ABB RobotStudio station: RemoteControlledYumi.rspag

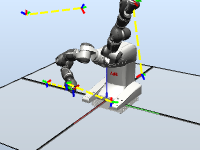
--- station ---
Station RemoteControlledYumi (saved by RobotStudio 6.5.7496.1049)
Controller IRB_14000_0.5kg_0.5m
  mechanical unit ROB_R: IRB14000_0.5_0.5_R, 6 joints, base frame (0, 0, 0) mm
  mechanical unit ROB_R_7: IRB14000_0.5_0.5_R, 1 joints, base frame (0, 0, 0) mm
  mechanical unit ROB_L: IRB14000_0.5_0.5_L, 6 joints, base frame (0, 0, 0) mm
  mechanical unit ROB_L_7: IRB14000_0.5_0.5_L, 1 joints, base frame (0, 0, 0) mm
Layout (positions relative to the parent item):
  - IRB14000_0.5_0.5 [mechanism, from Robots\IRB14000_0.5_0.5__01.rslib] at (0, 0, 0) mm
  - IRB14000_0.5_0.5_R [mechanism, from Robots\IRB14000_0.5_0.5__01.rslib] at (0, 0, 0) mm; joint values [1.0888, -1.6327, -1.6401, 0.7242, 2.6336, 0.3087, -2.7827] (rad or m)
  - IRB14000_0.5_0.5_L [mechanism, from Robots\IRB14000_0.5_0.5__01.rslib] at (0, 0, 0) mm; joint values [0.5159, -0.7237, 1.0056, -1.384, 2.6336, 0.3087, -2.7827] (rad or m)

--- Backups/IRB_14000_0.5kg_0.5m/RAPID/TASK1/PROGMOD/Module1.mod ---
MODULE Module1
	CONST jointtarget JointTarget_3:=[[5.435483871,-60.25483871,20.919354839,150.895790314,17.687340054,-159.437228739],[57.616129032,9E+09,9E+09,9E+09,9E+09,9E+09]];
	CONST jointtarget JointTarget_4:=[[29.560965021,-41.462551121,-79.294754901,150.895790314,17.687340054,-159.437228739],[57.616129032,9E+09,9E+09,9E+09,9E+09,9E+09]];
	CONST jointtarget JointTarget_1:=[[44.570967742,-88.003225806,2.538709677,0,39.999998836,0],[-79.358064516,9E+09,9E+09,9E+09,9E+09,9E+09]];
	CONST jointtarget JointTarget_2:=[[62.386456105,-93.54618891,41.493211378,150.895790314,17.687340054,-159.437228739],[-93.969401092,9E+09,9E+09,9E+09,9E+09,9E+09]];

    PROC main()
        RunLoop;
    ENDPROC
	PROC wavehigh()
	    MoveAbsJ JointTarget_3,v1000,fine,tool0\WObj:=wobj0;
	    MoveAbsJ JointTarget_4,v1000,z100,tool0\WObj:=wobj0;
	ENDPROC
	PROC wavelow()
	    MoveAbsJ JointTarget_1,v1000,z100,tool0\WObj:=wobj0;
	    MoveAbsJ JointTarget_2,v1000,z100,tool0\WObj:=wobj0;
	ENDPROC
ENDMODULE

--- Backups/IRB_14000_0.5kg_0.5m/RAPID/TASK1/PROGMOD/Remote.mod ---
MODULE Remote
    TASK PERS bool start := FALSE;
    TASK PERS bool running := FALSE;

    TASK PERS string name := "wavelow";

    PROC Init()
        start := FALSE;
        running := FALSE;
    ENDPROC

    PROC RunLoop()
        Init;
        WHILE TRUE DO
            WHILE NOT start DO
                WaitTime .1;
            ENDWHILE
            start := FALSE;
            running := TRUE;
            %name%;
            running := FALSE;
        ENDWHILE
    ENDPROC
ENDMODULE

--- Backups/IRB_14000_0.5kg_0.5m/RAPID/TASK1/SYSMOD/LINKEDM.sys ---
%%%
  VERSION:1
  LANGUAGE:ENGLISH
%%%

MODULE LINKEDM (SYSMODULE)

! FOLLOWER
!     Name of electronically linked follower axis used by operator at teach pendent.
      PERS string l_f_axis_name{5}       :=  ["",  "", "", "", ""];

!     Name of the mechanical unit for follower axis.
      PERS string l_f_mecunt_n{5}  :=  ["", "", "", "", ""];

!     Linked follower axis number in the mechanical unit (first axis in mech. unit is number 1).
      PERS num l_f_axis_no{5}      :=  [0,          0,   0,  0,  0];

! MASTER
!     Name of the mechanical unit for linked master axis.
      PERS string l_m_mecunt_n{5} :=  ["", "", "", "", ""];

!     Linked master axis number in the mechanical unit (first axis in mech. unit is number 1).
!     See axis number table in documentation for different master mechanical units.
      PERS num l_m_axis_no{5}     :=  [0,  0,  0,  0,  0];

! POSITION OFFSET
!     The increase of the allowed offset position between the master and follower
!     positions, used when starting AUTO mode. As soon as the offset is decreased
!     the old configurated parameter is used.
!     Example: 3 => the configurated value of allowed offset is increased 3 times.
      PERS num offset_ratio{5}       :=  [10,  10,   10,  10,  10];

! SPEED RATIO
!     Speed_ratio used in AUTO and JOG modes [ very_slow   slow    normal    fast]
!     Value 1 = max allowed manual speed.
      CONST num speed_ratio {20}      := [0.01, 0.01, 0.01, 0.01, 0.01,
                                          0.05, 0.05, 0.05, 0.05, 0.05,
                                          0.20, 0.20, 0.20, 0.20, 0.20,
                                          1.00, 1.00, 1.00, 1.00, 1.00];

! STEP SIZE
!     Displacement position used in JOG mode for each activation of positive or
!     negative movement.                  [very_short    short   normal   long]
!     Unit degees or meter.
      CONST num displacement {20}     := [0.001, 0.001, 0.001, 0.001, 0.001,
                                          0.005, 0.005, 0.005, 0.005, 0.005,
                                          0.020, 0.020, 0.020, 0.020, 0.020,
                                          0.100, 0.100, 0.100, 0.100, 0.100];


!-------------------------------------------------------------
 PROC Linked_m ()
      Linked_m_exe ;
 ENDPROC
ENDMODULE

--- Backups/IRB_14000_0.5kg_0.5m/RAPID/TASK2/PROGMOD/Module1.mod ---
MODULE Module1
	CONST jointtarget JointTarget_3:=[[5.435483871,-60.25483871,20.919354839,150.895790314,17.687340054,-159.437228739],[57.616129032,9E+09,9E+09,9E+09,9E+09,9E+09]];
	CONST jointtarget JointTarget_4:=[[29.560965021,-41.462551121,-79.294754901,150.895790314,17.687340054,-159.437228739],[57.616129032,9E+09,9E+09,9E+09,9E+09,9E+09]];
	CONST jointtarget JointTarget_1:=[[132.81046026,22.322183296,1.519468535,17.333519179,42.225247147,-11.8465977],[-86.991502251,9E+09,9E+09,9E+09,9E+09,9E+09]];
	CONST jointtarget JointTarget_2:=[[132.81046026,-30.727265036,-31.120707126,17.333519179,42.225247147,-11.8465977],[-86.991502251,9E+09,9E+09,9E+09,9E+09,9E+09]];

    PROC main()
        RunLoop;
    ENDPROC

	PROC wavehigh()
	    MoveAbsJ JointTarget_3,v1000,z100,tool0\WObj:=wobj0;
	    MoveAbsJ JointTarget_4,v1000,z100,tool0\WObj:=wobj0;
	ENDPROC

	PROC wavelow()
	    MoveAbsJ JointTarget_1,v1000,z100,tool0\WObj:=wobj0;
	    MoveAbsJ JointTarget_2,v1000,z100,tool0\WObj:=wobj0;
	ENDPROC
ENDMODULE

--- Backups/IRB_14000_0.5kg_0.5m/RAPID/TASK2/PROGMOD/Remote.mod ---
MODULE Remote
    TASK PERS bool start := FALSE;
    TASK PERS bool running := FALSE;

    TASK PERS string name := "wavehigh";

    PROC Init()
        start := FALSE;
        running := FALSE;
    ENDPROC

    PROC RunLoop()
        Init;
        WHILE TRUE DO
            WHILE NOT start DO
                WaitTime .1;
            ENDWHILE
            start := FALSE;
            running := TRUE;
            %name%;
            running := FALSE;
        ENDWHILE
    ENDPROC
ENDMODULE

--- Backups/IRB_14000_0.5kg_0.5m/SYSPAR/EIO.cfg ---
EIO:CFG_1.0:6:1::
#
SYSSIG_IN:

      -Signal "Collision_Avoidance" -Action "CollAvoidance"
#
INDUSTRIAL_NETWORK:

      -Name "EtherNetIP" -Connection "Private Network"\
      -Label "EtherNet/IP Adapter Network"

      -Name "DeviceNet" -Label "DeviceNet Master/Slave Network" -Address "2"
#
EIO_CROSS:

      -Name "Cross_Signal_Lamp" -Res "Signal_Lamp" -Act1 "DRV1BRAKE"
#
EIO_SIGNAL_SAFELEVEL:

      -Name "FlangePowerSafeLevel" -ActionWhenStartup "Last"
#
DEVICENET_DEVICE:

      -Name "D652_10" -VendorName "ABB Robotics" -ProductName "24 VDC Unit"\
      -Address 10 -ProductCode 26 -DeviceType 7 -ConnectionType "COS"\
      -OutputSize 2 -InputSize 2
#
DEVICENET_INTERNAL_DEVICE:

      -Name "DN_Internal_Device" -VendorName "ABB Robotics"\
      -ProductName "DeviceNet Internal Slave Device"
#
ETHERNETIP_INTERNAL_DEVICE:

      -Name "EN_Internal_Device" -VendorName "ABB Robotics"\
      -ProductName "EtherNet/IP Internal Adapter Device"
#
EIO_SIGNAL:

      -Name "custom_DI_0" -SignalType "DI" -Device "D652_10" -DeviceMap "0"

      -Name "custom_DI_1" -SignalType "DI" -Device "D652_10" -DeviceMap "1"

      -Name "custom_DI_2" -SignalType "DI" -Device "D652_10" -DeviceMap "2"

      -Name "custom_DI_3" -SignalType "DI" -Device "D652_10" -DeviceMap "3"

      -Name "custom_DI_4" -SignalType "DI" -Device "D652_10" -DeviceMap "4"

      -Name "custom_DI_5" -SignalType "DI" -Device "D652_10" -DeviceMap "5"

      -Name "custom_DI_6" -SignalType "DI" -Device "D652_10" -DeviceMap "6"

      -Name "custom_DI_7" -SignalType "DI" -Device "D652_10" -DeviceMap "7"

      -Name "custom_DO_0" -SignalType "DO" -Device "D652_10" -DeviceMap "0"

      -Name "custom_DO_1" -SignalType "DO" -Device "D652_10" -DeviceMap "1"

      -Name "custom_DO_2" -SignalType "DO" -Device "D652_10" -DeviceMap "2"

      -Name "custom_DO_3" -SignalType "DO" -Device "D652_10" -DeviceMap "3"

      -Name "custom_DO_4" -SignalType "DO" -Device "D652_10" -DeviceMap "4"

      -Name "custom_DO_5" -SignalType "DO" -Device "D652_10" -DeviceMap "5"

      -Name "custom_DO_6" -SignalType "DO" -Device "D652_10" -DeviceMap "6"

      -Name "custom_DO_7" -SignalType "DO" -Device "D652_10" -DeviceMap "7"

      -Name "hall_sensor_joint_1" -SignalType "DI" -Device "D652_10"\
      -DeviceMap "8"

      -Name "hall_sensor_joint_2" -SignalType "DI" -Device "D652_10"\
      -DeviceMap "9"

      -Name "hall_sensor_joint_3" -SignalType "DI" -Device "D652_10"\
      -DeviceMap "11"

      -Name "hall_sensor_joint_4" -SignalType "DI" -Device "D652_10"\
      -DeviceMap "12"

      -Name "hall_sensor_joint_5" -SignalType "DI" -Device "D652_10"\
      -DeviceMap "13"

      -Name "hall_sensor_joint_6" -SignalType "DI" -Device "D652_10"\
      -DeviceMap "14"

      -Name "hall_sensor_joint_7" -SignalType "DI" -Device "D652_10"\
      -DeviceMap "10"

      -Name "hall_sensor_24V_ROB_R" -SignalType "DO" -Device "D652_10"\
      -DeviceMap "8"

      -Name "hall_sensor_24V_ROB_L" -SignalType "DO" -Device "D652_10"\
      -DeviceMap "9"

      -Name "flange_24V_ROB_R" -SignalType "DO" -Device "D652_10"\
      -DeviceMap "10" -SafeLevel "FlangePowerSafeLevel"

      -Name "flange_24V_ROB_L" -SignalType "DO" -Device "D652_10"\
      -DeviceMap "11" -SafeLevel "FlangePowerSafeLevel"

      -Name "Signal_Lamp" -SignalType "DO" -Device "D652_10" -DeviceMap "12"

      -Name "Collision_Avoidance" -SignalType "DO" -Access "All" -Default 1
